# EPICS substitutions: evrSupport/Db/ioc/IOC-IN20-RF01pattern.substitutions
#
# Pattern records
file evrPattern.template {
#	    Device        ,  SLC Pattern Check LNK    , EVR/Trigger
#	                                                  Links
  pattern { DEVICE        ,        LINK4              , LINK5 , LINK6 , LINKD }
	  { IOC:IN20:RF01 ,         ""                ,  ""   ,  ""   ,  ""   }
}
file evrPatternProc.template {
  pattern { DEVICE }
	  { IOC:IN20:RF01}
}
